# EPICS autosave request: ipApp/Db/SRS_SG390_settings.req
$(P)$(R):readAll.SCAN
$(P)$(R):freq.VAL
$(P)$(R):freqMHz.VAL
$(P)$(R):amp.VAL
$(P)$(R):ampRMS.VAL
$(P)$(R):phase.VAL
$(P)$(R):rf.VAL
$(P)$(R):lf.VAL
$(P)$(R):freq.PREC
$(P)$(R):freqMHz.PREC
$(P)$(R):amp.PREC
$(P)$(R):ampRMS.PREC
$(P)$(R):phase.PREC
$(P)$(R):freq_RBV.PREC
$(P)$(R):freqMHz_RBV.PREC
$(P)$(R):amp_RBV.PREC
$(P)$(R):ampRMS_RBV.PREC
$(P)$(R):phase_RBV.PREC
